PROGRAM MAIN_Sender
VAR
	// SMPTE Time Controller
	SMPTE_TimeController : FB_SMPTE_TimeController(eTimeSource := E_SMPTE_TimeController_Source.ExtTimeProvider, eFrameMode := E_SMPTE_FrameMode.FPS_25);
	// SMPTE Sender
	SMPTE_Sender 	: FB_SMPTE_Sender(ipSMPTE_TimeController := SMPTE_TimeController);
	
	// External Time Source
	nSysTime AT %I* : ULINT;
	
	// Enable the sender
	bEnableSending: BOOL;
	// Disable the sender
	bDisableSending: BOOL;
	// Error status of sender
	bSMPTE_Error: BOOL;
	// Enable Status
	bSMPTE_Enabled: BOOL;
	
	// Play the timeline
	bPlay: BOOL;
	// Pause the timeline
	bPause: BOOL;
	// Stop the timeline
	bStop: BOOL;
	// Reset the timeline
	bReset: BOOL;
	
	// View the current time struct being send
	stSMPTE_TimeStruct : ST_SMPTE_TimeStruct;

END_VAR

(**********************)
(**** SMPTE Sender ****)
(**********************)

// Call once each cycle
SMPTE_TimeController.Cycle();
SMPTE_Sender.Cycle();

// Enable sending the SMPTE signal
IF SMPTE_Sender.EnableSending(bExecute := bEnableSending) THEN
	bEnableSending := FALSE;
END_IF

// Disable sending the SMPTE signal
IF SMPTE_Sender.DisableSending(bExecute := bDisableSending) THEN
	bDisableSending := FALSE;
END_IF

// Check if errors on SMPTE Sender
bSMPTE_Error := SMPTE_Sender.Error;
// Check if enabled
bSMPTE_Enabled := SMPTE_Sender.Enabled;



(********************************)
(**** SMPTE Time Conectoller ****)
(********************************)

// Assign External Time Source
SMPTE_TimeController.AssignExternalTimeSource(nSysTime);

// Playback controls
IF SMPTE_TimeController.Play(bExecute := bPlay) THEN
	bPlay := FALSE;
END_IF

IF SMPTE_TimeController.Pause(bExecute := bPause) THEN
	bPause := FALSE;
END_IF

IF SMPTE_TimeController.Stop(bExecute := bStop) THEN
	bStop := FALSE;
END_IF

IF SMPTE_TimeController.Reset(bExecute := bReset) THEN
	bReset := FALSE;
END_IF

// Sample of Timecode being send
stSMPTE_TimeStruct := SMPTE_TimeController.TimeStruct;

END_PROGRAM

(* stored: Version 1.1.0.1, ProductVersion 3.1.4024.12
   POU MAIN_Sender: Id {83453181-9632-4c50-a095-465548438677}, SpecialFunc None *)
